TYPE ST_TrayLayerPositionConfig :
STRUCT
    fHighPosition : LREAL;
    fLowPosition : LREAL;
END_STRUCT
END_TYPE

(* stored: Version 1.1.0.1, ProductVersion 3.1.4026.20
   DUT ST_TrayLayerPositionConfig: Id {1a53ff19-47bd-4f6f-8a3a-1591d1870c17} *)
